TYPE ST_ParaVal_UpdateVise :
STRUCT
	ViseNumber			: SINT;
	SerialNumber		: STRING(255);
	DutIdentifier		: LINT;
	CamIdentifier		: LINT;
	CncNumber			: SINT;
END_STRUCT
END_TYPE

(* stored: Version 1.1.0.1, ProductVersion 3.1.4024.11
   DUT ST_ParaVal_UpdateVise: Id {4d615083-e16e-4560-9f94-a0c07b3168fe} *)
